SYSTEM System (* System Configuration *)
  (* Standard: 61499-1 *)
  (* Version 0.0, 18/05/2022, Admin, Schneider Electric *)
  {SET_ATTRIBUTE(System.Device.FolderPath, EcoRT_0,DEV)}
  APPLICATION APP1
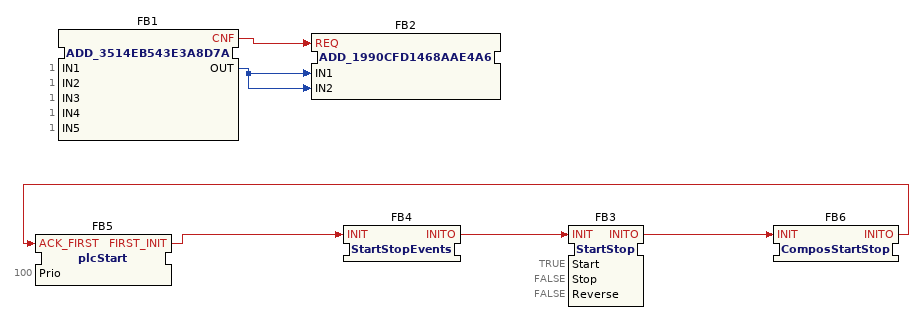
    FBS
      FB1 : ADD_3514EB543E3A8D7A(IN1 := 1, IN2 := 1, IN3 := 1, IN4 := 1, IN5 := 1); {SET_ATTRIBUTE(Configuration.GenericFBType.InterfaceParams, Runtime.Standard#CNT:=5;IN${CNT$}:INT)}
      FB2 : ADD_1990CFD1468AAE4A6; {SET_ATTRIBUTE(Configuration.GenericFBType.InterfaceParams, Runtime.Standard#CNT:=2;IN${CNT$}:LREAL)}
      FB3 : StartStop(Start := TRUE, Stop := FALSE, Reverse := FALSE);
      FB4 : StartStopEvents;
      FB5 : plcStart(Prio := 100);
      FB6 : ComposStartStop;
    END_FBS
    EVENT_CONNECTIONS
      FB1.CNF TO FB2.REQ;
      FB5.FIRST_INIT TO FB4.INIT;
      FB4.INITO TO FB3.INIT;
      FB3.INITO TO FB6.INIT;
      FB6.INITO TO FB5.ACK_FIRST;
    END_CONNECTIONS
    DATA_CONNECTIONS
      FB1.OUT TO FB2.IN1;
      FB1.OUT TO FB2.IN2;
    END_CONNECTIONS
  END_APPLICATION
  DEVICE EcoRT_0 : Soft_dPAC
    RESOURCE RES0 : EMB_RES_ECO
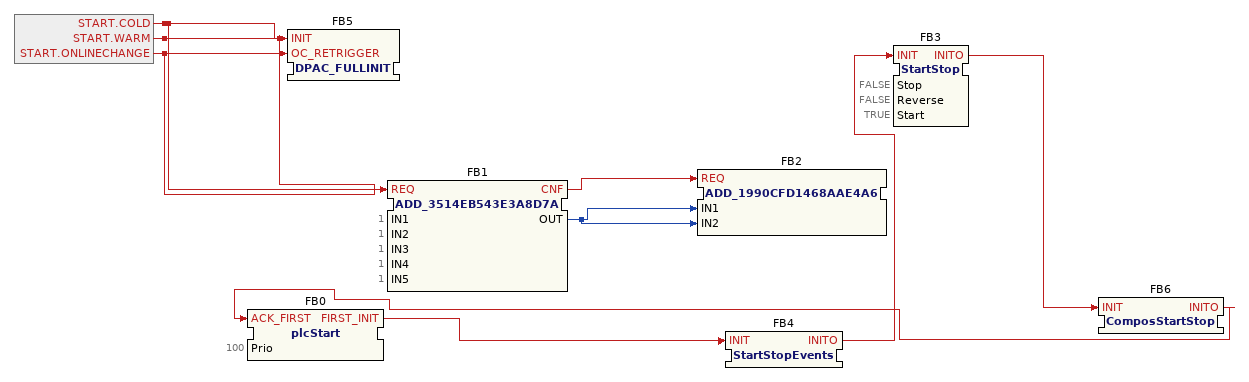
      FBS
        FB1 : ADD_3514EB543E3A8D7A(IN1 := 1, IN2 := 1, IN3 := 1, IN4 := 1, IN5 := 1); {SET_ATTRIBUTE(Configuration.GenericFBType.InterfaceParams, Runtime.Standard#CNT:=5;IN${CNT$}:INT)}
        FB2 : ADD_1990CFD1468AAE4A6; {SET_ATTRIBUTE(Configuration.GenericFBType.InterfaceParams, Runtime.Standard#CNT:=2;IN${CNT$}:LREAL)}
        FB4 : StartStopEvents;
        FB3 : StartStop(Stop := FALSE, Reverse := FALSE, Start := TRUE);
        FB5 : DPAC_FULLINIT;
        FB0 : plcStart(Prio := 100);
        FB6 : ComposStartStop;
      END_FBS
      EVENT_CONNECTIONS
        START.COLD TO FB1.REQ;
        START.WARM TO FB1.REQ;
        START.ONLINECHANGE TO FB1.REQ;
        FB1.CNF TO FB2.REQ;
        START.COLD TO FB5.INIT;
        START.WARM TO FB5.INIT;
        START.ONLINECHANGE TO FB5.OC_RETRIGGER;
        FB4.INITO TO FB3.INIT;
        FB0.FIRST_INIT TO FB4.INIT;
        FB3.INITO TO FB6.INIT;
        FB6.INITO TO FB0.ACK_FIRST;
      END_CONNECTIONS
      DATA_CONNECTIONS
        FB1.OUT TO FB2.IN1;
        FB1.OUT TO FB2.IN2;
      END_CONNECTIONS
    END_RESOURCE
  END_DEVICE
  DEVICE DEV : M580_dPAC
    RESOURCE RES0 : EMB_RES_ECO
    END_RESOURCE
  END_DEVICE
  MAPPINGS
    APP1.FB1 ON EcoRT_0.RES0;
    APP1.FB2 ON EcoRT_0.RES0;
    APP1.FB4 ON EcoRT_0.RES0;
    APP1.FB3 ON EcoRT_0.RES0;
    APP1.FB5 ON EcoRT_0.RES0.FB0;
    APP1.FB6 ON EcoRT_0.RES0;
  END_MAPPINGS
END_SYSTEM
